PROGRAM MAIN
VAR
	Alarms : AlarmServer;	
	Berra: BOOL;
	Baz: BOOL;
	Ack: BOOL;
	clear: BOOL;
	ddd: BOOL;
	
	startTime			: ULINT;
	stopTime			: ULINT;
	diffTime			: ULINT;
	i :INT;	
	AckAll: BOOL;
	READ: BOOL;

	number: INT := 5;
END_VAR

Alarms();

IF Berra THEN
	startTime:= F_GetActualDcTime64();
	Berra := FALSE;
		
	FOR i:=0 TO number DO 
		Alarms.NewAlarm(sName:=INT_TO_STRING(i), sAlarmText:= 'Ett nytt larm');
	END_FOR
	
	stopTime:= F_GetActualDcTime64();
	diffTime := (stopTime - startTime);
END_IF
IF Baz THEN
	Baz := FALSE;
		
	Alarms.NewAlarm(sName:='Bingo', sAlarmText:= 'Ett nytt larm');
	Alarms.NewAlarm(sName:='Baz', sAlarmText:= 'Ett nytt larm');
	Alarms.NewAlarm(sName:='Tjo', sAlarmText:= 'Ett nytt larm');
	Alarms.NewAlarm(sName:='Tjo', sAlarmText:= 'Bazinga');
END_IF


IF Ack THEN
	startTime:= F_GetActualDcTime64();
	Ack := FALSE;
	Alarms.AckAlarm(iRow:= 900 );
	stopTime:= F_GetActualDcTime64();
	diffTime := (stopTime - startTime);
END_IF

IF AckAll THEN
	startTime:= F_GetActualDcTime64();
	AckAll := FALSE;
	Alarms.AckAllAlarms();
	stopTime:= F_GetActualDcTime64();
	diffTime := (stopTime - startTime);
END_IF

IF clear THEN
	clear := FALSE;
	Alarms.ClearAllAlarms();
END_IF

IF ddd THEN
	ddd := FALSE;
		
	Alarms.NewAlarm(sName:='Braf', sAlarmText:= 'Ett nytt larm');
	Alarms.NewAlarm(sName:='Gizmo', sAlarmText:= 'Ett nytt larm');
END_IF

IF READ THEN
	startTime:= F_GetActualDcTime64();
	READ := FALSE;
	Alarms.ReadFromDB(NrOfRows:= 10);
	stopTime:= F_GetActualDcTime64();
	diffTime := (stopTime - startTime);
END_IF

END_PROGRAM

(* stored: Version 1.1.0.1, ProductVersion 3.1.4024.9
   POU MAIN: Id {9a484491-9707-4649-bff0-788e52f873b2}, SpecialFunc None *)
